{attribute addProperty BoxType "EL4732-0001-0000"}
{attribute addProperty Id "Cycle_CounterAT %Q*Cycle_Counter_485675001620Sample_0AT %Q*Sample_6DB94BDA3240WcStateAT %I*WcState_28A8677510.1250InfoDataAT %I*InfoData_7231B2DD80100"}
{attribute addProperty CRC "456969579"}
{attribute addProperty SizeInBites "129"}
{attribute addProperty SizeInBytes "16.125"}
TYPE EL4732_A4B0F6DE :
STRUCT
	{attribute addProperty Name "Cycle_Counter"}
	Cycle_Counter : Cycle_Counter_48567500;
	{attribute addProperty Name "Sample_0"}
	Sample_0 : Sample_6DB94BDA;
	{attribute addProperty Name "WcState"}
	WcState : WcState_28A86775;
	{attribute addProperty Name "InfoData"}
	InfoData : InfoData_7231B2DD;
END_STRUCT
END_TYPE

(* stored: Version 1.2.0.0, ProductVersion 3.1.4024.9
   DUT EL4732_A4B0F6DE: Id {f49af053-f55e-441c-bc6b-b8a79f4dd4d6} *)
